Fanuc TP program (LS listing): UP201.LS

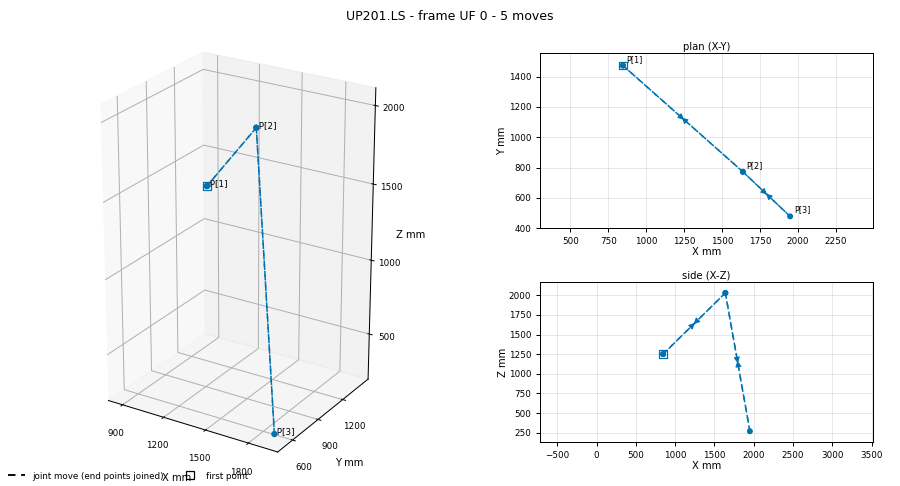
[picture p0: tool path of UP201.LS in frame UF 0, 5 of 5 moves have a stored position in this frame; points joined in program order, loops and branches not executed]
/PROG  UP201
/ATTR
OWNER		= AUROM;
COMMENT		= "Camb. Herr. G1";
PROG_SIZE	= 2712;
CREATE		= DATE 03-15-00  TIME 13:37:40;
MODIFIED	= DATE 16-11-27  TIME 00:48:48;
FILE_NAME	= ;
VERSION		= 0;
LINE_COUNT	= 9;
MEMORY_SIZE	= 4780;
PROTECT		= READ_WRITE;
TCD:  STACK_SIZE	= 500,
      TASK_PRIORITY	= 50,
      TIME_SLICE	= 0,
      BUSY_LAMP_OFF	= 0,
      ABORT_REQUEST	= 0,
      PAUSE_REQUEST	= 0;
DEFAULT_GROUP	= 1,1,1,1,*;
CONTROL_CODE	= 00000000 00000000;
/MN
   1:  UTOOL_NUM=1 ;
   2:  UFRAME_NUM=0 ;
   3:  PAYLOAD[1] ;
   4:J P[1] 100% CNT0 ACC100 TB    .10sec,P-SPS    ;
      1:  TC_ONLINE (ON) ;
      2:  DO[23]=OFF ;
      3:  CALL MAKRO050    ;
      4:  !Lib. de Herramientas ;
      5:  DO[80]=ON ;
      6:  DO[78]=OFF ;
      7:  DO[77]=ON ;
      8:  DO[75]=OFF ;
      9:  DO[74]=ON ;
     10:  DO[73]=ON ;
     11:  DO[72]=OFF ;
     12:  DO[71]=OFF ;
     13:  DO[69]=OFF ;
     14:  !Lib. de Anticolisiones ;
     15:  DO[41]=ON ;
     16:  DO[42]=ON ;
     17:  DO[43]=ON ;
     18:  DO[44]=ON ;
     19:  DO[45]=ON ;
     20:  DO[46]=ON ;
     21:  !Apagar Pos. Base ;
     22:  DO[15]=OFF ;
     23:  !Robot en Trayectoria ;
     24:  DO[16]=ON ;
     25:  WAIT (DI[23])    ;
     26:  DO[23]=ON ;
     27:  TC_ONLINE (M[2] AND M[30] AND M[31] AND M[33] AND M[35] AND M[37] AND M[39] AND M[41] AND M[95] AND M[96]) ;
       ------ ;
   5:J P[2] 100% CNT100 ACC100 TB   0.00sec,P-SPS    ;
      1:  TC_ONLINE (M[2] AND M[30] AND M[31] AND M[33] AND M[35] AND M[37] AND M[39] AND M[41] AND M[95] AND M[96]) ;
       ------ ;
   6:  !Cambio de Herramienta ;
   7:J P[3] 100% CNT0 ACC100 TB    .10sec,P-SPS    ;
      1:  TC_ONLINE (ON) ;
      2:  DO[23]=OFF ;
      3:  DO[17]=ON ;
      4:  GO[19]=1 ;
      5:  WAIT (DI[17])    ;
      6:  DO[17]=OFF ;
      7:  GO[19]=0 ;
      8:  WAIT (DI[23])    ;
      9:  DO[23]=ON ;
     10:  TC_ONLINE (M[2] AND M[30] AND M[31] AND M[33] AND M[35] AND M[37] AND M[39] AND M[41] AND M[95] AND M[96]) ;
       ------ ;
   8:J P[4] 100% CNT100 ACC100 TB   0.00sec,P-SPS    ;
      1:  TC_ONLINE (M[2] AND M[30] AND M[31] AND M[33] AND M[35] AND M[37] AND M[39] AND M[41] AND M[95] AND M[96]) ;
       ------ ;
   9:J P[5] 100% CNT0 ACC100 TB    .10sec,P-SPS    ;
      1:  TC_ONLINE (ON) ;
      2:  DO[23]=OFF ;
      3:  WAIT (DI[23])    ;
      4:  DO[23]=ON ;
      5:  TC_ONLINE (M[2] AND M[30] AND M[31] AND M[33] AND M[35] AND M[37] AND M[39] AND M[41] AND M[95] AND M[96]) ;
       ------ ;
/POS
P[1]{
   GP1:
	UF : 0, UT : 1,		CONFIG : 'N U T, 0, 0, 0',
	X =   846.483  mm,	Y =  1473.446  mm,	Z =  1251.233  mm,
	W =   -40.712 deg,	P =    36.105 deg,	R =    90.967 deg
   GP2:
	UF : 0, UT : 1,
	J1=   100.000  mm
   GP3:
	UF : 0, UT : 1,
	J1=     0.000  mm
   GP4:
	UF : 0, UT : 1,
	J1=     0.000  mm
};
P[2]{
   GP1:
	UF : 0, UT : 1,		CONFIG : 'N U T, 0, 0, 0',
	X =  1638.382  mm,	Y =   772.101  mm,	Z =  2029.092  mm,
	W =   -85.756 deg,	P =     1.670 deg,	R =    42.112 deg
   GP2:
	UF : 0, UT : 1,
	J1=   100.000  mm
   GP3:
	UF : 0, UT : 1,
	J1=     0.000  mm
   GP4:
	UF : 0, UT : 1,
	J1=     0.000  mm
};
P[3]{
   GP1:
	UF : 0, UT : 1,		CONFIG : 'F U T, 0, 0, 0',
	X =  1950.086  mm,	Y =   477.852  mm,	Z =   270.228  mm,
	W =   -91.167 deg,	P =    -3.743 deg,	R =    33.700 deg
   GP2:
	UF : 0, UT : 1,
	J1=   100.000  mm
   GP3:
	UF : 0, UT : 1,
	J1=     0.000  mm
   GP4:
	UF : 0, UT : 1,
	J1=     0.000  mm
};
P[4]{
   GP1:
	UF : 0, UT : 1,		CONFIG : 'N U T, 0, 0, 0',
	X =  1638.382  mm,	Y =   772.101  mm,	Z =  2029.092  mm,
	W =   -85.756 deg,	P =     1.670 deg,	R =    42.112 deg
   GP2:
	UF : 0, UT : 1,
	J1=   100.000  mm
   GP3:
	UF : 0, UT : 1,
	J1=     0.000  mm
   GP4:
	UF : 0, UT : 1,
	J1=     0.000  mm
};
P[5]{
   GP1:
	UF : 0, UT : 1,		CONFIG : 'N U T, 0, 0, 0',
	X =   846.483  mm,	Y =  1473.446  mm,	Z =  1251.233  mm,
	W =   -40.712 deg,	P =    36.105 deg,	R =    90.967 deg
   GP2:
	UF : 0, UT : 1,
	J1=   100.000  mm
   GP3:
	UF : 0, UT : 1,
	J1=     0.000  mm
   GP4:
	UF : 0, UT : 1,
	J1=     0.000  mm
};
/END
